PROGRAM Delta
VAR
END_VAR

GVL.astAxes[AXIS_DELTA].stInputs.bLimitBwd := TRUE;
GVL.astAxes[AXIS_DELTA].stInputs.bLimitFwd := TRUE;
GVL.astAxes[AXIS_DELTA].stControl.bEnable := TRUE;

astAxes[AXIS_DELTA].stDescription.sAxisName := 'DELTA';

END_PROGRAM

(* stored: Version 1.1.0.1, ProductVersion 3.1.4024.12
   POU Delta: Id {327f0294-cf79-49cf-a462-33ee499ace55}, SpecialFunc None *)
